{attribute 'qualified_only'}
VAR_GLOBAL
	g_xSimulationActive :BOOL :=TRUE;
	Timerlong : TON;
	TimerShort : TON;
END_VAR

(* stored: Version 1.1.0.1
   GVL GVL: Id {46730589-20a3-41d6-acda-4d560c7a530e} *)
